FUNCTION_BLOCK FB_GantryAutoCoupling_Test EXTENDS TcUnit.FB_TestSuite
VAR
    Expected: BOOL;
    Actual: BOOL;
END_VAR

TEST('FB_GantryAutoCoupling_Test Dummy Test');
AssertEquals(Expected := Expected,
             Actual := Actual,
             Message := 'Error Message');
TEST_FINISHED();

END_FUNCTION_BLOCK

(* stored: Version 1.1.0.1, ProductVersion 3.1.4022.18
   POU FB_GantryAutoCoupling_Test: Id {4f3e0252-75d1-4b0c-b8b2-c0af48301fa0}, SpecialFunc None *)
